TYPE ST_Bleutooth :
STRUCT
	Status AT%I*	: ST_Bleutooth_Status	; // status inputs
	control AT%Q*	: ST_BleutoothControl	; // Control Outputs
END_STRUCT
END_TYPE

(* stored: Version 1.1.0.1
   DUT ST_Bleutooth: Id {f86b691b-ec88-418e-99da-da89b35f53ba} *)
